// TIA Portal V20 export
TYPE "type_emRelations_em13_cmStatus"
// stored: Access Published, Namespace Unit1
   STRUCT
      JRUnloadingPnPSafetyPin : "LBC_typeDigitalSignalControlNode";
      JRUnloadingPnPJRDetect : "LBC_typeDigitalSignalControlNode";
      JRUnloadingPnPAxisX : "LBC_typeAxis64PosControlNode";
      JRUnloadingPnPAxisZ : "LBC_typeAxis64PosControlNode";
      JRUnloadingPnPAxisC : "LBC_typeAxis64PosControlNode";
      JRUnloadingPnPClampOpenClose : "LBC_typeTwoWayActuatorControlNode";
   END_STRUCT;
END_TYPE
